(* Single tank with LimitSwitchLow (piLsLow) and LimitSwitchHigh (piLsHigh)
| using this function when have to DEPENDENT Measure weight
*)
FUNCTION_BLOCK FB_SingleTankV0 EXTENDS FB_SingleTank
VAR
	bAllowInMaterial : BOOL;
	bAllowOutMaterial : BOOL;
	tonRemainOffLsLow	: TON;
	tRemainOffLsLow	: TIME := T#1S;
	tonRemainLsHigh	: TON;
	tRemainLsHigh	: TIME := T#1S;	
END_VAR

tonRemainOffLsLow(
	IN := NOT piLslow.In,
	PT := tRemainOffLsLow,
);
bAllowOutMaterial := NOT tonRemainOffLsLow.Q;

tonRemainLsHigh(
	IN := piLsHigh.In,
	PT := tRemainLsHigh,
);
bAllowInMaterial := NOT tonRemainLsHigh.Q;
SUPER^();

PROPERTY AllowIn : Reference to bool
GET
AllowIn ref= bAllowInMaterial;
END_GET
END_PROPERTY

(*
| Check the minimum condition  (lrWeight > lrLimitMinWeight
								AND piLslow.In;)
*)
PROPERTY AllowOut : REFERENCE TO BOOL
GET
AllowOut ref= bAllowOutMaterial;
END_GET
END_PROPERTY

PROPERTY TimeRemainLsHigh : Time
GET
TimeRemainLsHigh := tRemainLsHigh;
END_GET
SET
tRemainLsHigh := TimeRemainLsHigh;
END_SET
END_PROPERTY

PROPERTY TimeRemainOffLsLow : Time
GET
TimeRemainOffLsLow := tRemainOffLsLow;
END_GET
SET
tRemainOffLsLow := TimeRemainOffLsLow;
END_SET
END_PROPERTY

END_FUNCTION_BLOCK

(* stored: Version 1.1.0.1, ProductVersion 3.1.4024.12
   POU FB_SingleTankV0: Id {804ff059-bff6-46a3-be72-e0e118682176}, SpecialFunc None
   Property AllowIn: Id {fc712f05-a064-4a5a-96e7-72aaec14e8cf}
   Get Get: Id {5c729add-9dbd-4aa3-b258-be82a8761357}
   Property AllowOut: Id {0e0965dc-bf3f-4465-bfeb-792393b01443}
   Get Get: Id {b01519fc-927a-40ec-ba86-a2b2d4e2c6ab}
   Property TimeRemainLsHigh: Id {d11668c1-4f5e-40de-b8e3-d91045ad5ba3}
   Get Get: Id {b2101392-74b9-4f15-b14e-856ba87f9441}
   Set Set: Id {a8dcedc0-952b-4dfd-8752-ce18e8877301}
   Property TimeRemainOffLsLow: Id {64cb247d-190a-47c7-ad90-c3b9b3de1b1f}
   Get Get: Id {90f07dfc-6052-4ae2-979f-1e568ca273d6}
   Set Set: Id {b31d19b4-b14d-4e81-81c5-713e73b41b0c} *)
